// TIA Portal V20 export
TYPE "type_emRelations_em4_sequence"
// stored: Access Published, Namespace Unit1
   STRUCT
      sideTapeLoading : Struct
         jobs : "LAF_typeJobs";
         sequence : "LAF_typeSequence";
         selectJobStatus { S7_SetPoint := 'True'} : Array[0..10] of "LAF_typeJobStatus";
         "step" : "LER_typeStep";
         jobInterface : Struct
            chargeJob2 : "LER_typeJobInterface";
         END_STRUCT;
         homeCheck : Struct
            TapeLoadReq { ExternalWritable := 'False'} : Bool;
            TapeLoaded { ExternalWritable := 'False'} : Bool;
         END_STRUCT;
      END_STRUCT;
      sideTapeAttachment : Struct
         jobs : "LAF_typeJobs";
         sequence : "LAF_typeSequence";
         selectJobStatus { S7_SetPoint := 'True'} : Array[0..10] of "LAF_typeJobStatus";
         "step" : "LER_typeStep";
         jobInterface : Struct
            rightTapeGetJob2 : "LER_typeJobInterface";
            leftTapeGetJob3 : "LER_typeJobInterface";
            tape1PutJob4 : "LER_typeJobInterface";
            tape2PutJob5 : "LER_typeJobInterface";
            tape3PutJob6 : "LER_typeJobInterface";
            tape4PutJob7 : "LER_typeJobInterface";
            TapeIdleJob8 { S7_SetPoint := 'True'} : "LER_typeJobInterface";
         END_STRUCT;
         homeCheck : Struct
            waitPosTapeGetReq { ExternalWritable := 'False'} : Bool;
            waitPosTapeLeftGet { ExternalWritable := 'False'} : Bool;
            waitPosTapeRightGet { ExternalWritable := 'False'} : Bool;
            waitPosTapeAllGet { ExternalWritable := 'False'} : Bool;
            putPosTapeAllGet { ExternalWritable := 'False'} : Bool;
         END_STRUCT;
      END_STRUCT;
      sideTapeFixStage : Struct
         jobs : "LAF_typeJobs";
         sequence : "LAF_typeSequence";
         selectJobStatus { S7_SetPoint := 'True'} : Array[0..10] of "LAF_typeJobStatus";
         "step" : "LER_typeStep";
         jobInterface : Struct
            loadJob2 : "LER_typeJobInterface";
            taping1Job3 : "LER_typeJobInterface";
            taping2Job4 : "LER_typeJobInterface";
            taping3Job5 : "LER_typeJobInterface";
            taping4Job6 : "LER_typeJobInterface";
            unloadJob7 : "LER_typeJobInterface";
         END_STRUCT;
         homeCheck : Struct
            tape1PosPartNoDetect { ExternalWritable := 'False'} : Bool;
            tape1PosPartDetect { ExternalWritable := 'False'} : Bool;
            tape2PosPartDetect { ExternalWritable := 'False'} : Bool;
            tape3PosPartDetect { ExternalWritable := 'False'} : Bool;
            tape4PosPartDetect { ExternalWritable := 'False'} : Bool;
         END_STRUCT;
      END_STRUCT;
   END_STRUCT;
   // // sideTapeLoading."step".action1[101] : Step[101] : JOB[1] Condition
   // // sideTapeLoading."step".action1[110] : Step[110] : Side Tape Loading Down
   // // sideTapeLoading."step".action1[120] : Step[120] : Side Tape Clamp Open
   // // sideTapeLoading."step".action1[130] : Step[130] : Side Tape Cutter Backward
   // // sideTapeLoading."step".action1[140] : Step[140] : Side Tape Cutter Clamp Forward
   // // sideTapeLoading."step".action1[150] : Step[150] : Side Tape Tension Backward
   // // sideTapeLoading."step".action1[190] : Step[190] : JOB[1] Step End
   // // sideTapeLoading."step".action1[201] : Step[201] : JOB[2] Condition
   // // sideTapeLoading."step".action1[210] : Step[210] : Side Tape Loading Up, Tension Backward
   // // sideTapeLoading."step".action1[220] : Step[220] : Side Tape Clamp Close
   // // sideTapeLoading."step".action1[230] : Step[230] : Side Tape Cutter Clamp Backward
   // // sideTapeLoading."step".action1[240] : Step[240] : Side Tape Loading Down, Tension Forward
   // // sideTapeLoading."step".action1[250] : Step[250] : Side Tape Cutter Clamp Forward
   // // sideTapeLoading."step".action1[260] : Step[260] : Side Tape Tension Backward
   // // sideTapeLoading."step".action1[290] : Step[290] : JOB[2] Step End
   // // sideTapeLoading."step".transition1[101] : Step[101] : JOB[1] Condition
   // // sideTapeLoading."step".transition1[110] : Step[110] : Side Tape Loading Down
   // // sideTapeLoading."step".transition1[120] : Step[120] : Side Tape Clamp Open
   // // sideTapeLoading."step".transition1[130] : Step[130] : Side Tape Cutter Backward
   // // sideTapeLoading."step".transition1[140] : Step[140] : Side Tape Cutter Clamp Forward
   // // sideTapeLoading."step".transition1[150] : Step[150] : Side Tape Tension Backward
   // // sideTapeLoading."step".transition1[190] : Step[190] : JOB[1] Step End
   // // sideTapeLoading."step".transition1[201] : Step[201] : JOB[2] Condition
   // // sideTapeLoading."step".transition1[210] : Step[210] : Side Tape Loading Up, Tension Backward
   // // sideTapeLoading."step".transition1[220] : Step[220] : Side Tape Clamp Close
   // // sideTapeLoading."step".transition1[230] : Step[230] : Side Tape Cutter Clamp Backward
   // // sideTapeLoading."step".transition1[240] : Step[240] : Side Tape Loading Down, Tension Forward
   // // sideTapeLoading."step".transition1[250] : Step[250] : Side Tape Cutter Clamp Forward
   // // sideTapeLoading."step".transition1[260] : Step[260] : Side Tape Tension Backward
   // // sideTapeLoading."step".transition1[290] : Step[290] : JOB[2] Step End
   // // sideTapeAttachment."step".action1[101] : Step[101] : JOB[1] Condition
   // // sideTapeAttachment."step".action1[110] : Step[110] : Side Tape Attachment Left, Right Backward
   // // sideTapeAttachment."step".action1[111] : Step[111] : Side Tape Attachment Y-Axis Wait Pos
   // // sideTapeAttachment."step".action1[120] : Step[120] : Side Tape Attachment Bottom Forward
   // // sideTapeAttachment."step".action1[130] : Step[130] : Side Tape Attachment Remain Attach Left Condition
   // // sideTapeAttachment."step".action1[131] : Step[131] : Side Tape Attachment X-Axis Remain Attach Left Position
   // // sideTapeAttachment."step".action1[132] : Step[132] : Side Tape Attachment Y-Axis Remain Attach Left Position
   // // sideTapeAttachment."step".action1[133] : Step[133] : Side Tape Attachment Left Vaccum Off
   // // sideTapeAttachment."step".action1[134] : Step[134] : Side Tape Attachment Y-Axis Wait Pos
   // // sideTapeAttachment."step".action1[140] : Step[140] : Side Tape Attachment Remain Attach Right Condition
   // // sideTapeAttachment."step".action1[141] : Step[141] : Side Tape Attachment X-Axis Remain Attach Right Position
   // // sideTapeAttachment."step".action1[142] : Step[142] : Side Tape Attachment Y-Axis Remain Attach Right Position
   // // sideTapeAttachment."step".action1[143] : Step[143] : Side Tape Attachment Right Vaccum Off
   // // sideTapeAttachment."step".action1[144] : Step[144] : Side Tape Attachment Y-Axis Wait Pos
   // // sideTapeAttachment."step".action1[180] : Step[180] : Side Tape Attachment X-Axis Wait Position
   // // sideTapeAttachment."step".action1[190] : Step[190] : Job[1] Step End
   // // sideTapeAttachment."step".action1[201] : Step[201] : JOB[2] Condition
   // // sideTapeAttachment."step".action1[210] : Step[210] : Side Tape Attachment X-Axis Right Loading Pos
   // // sideTapeAttachment."step".action1[220] : Step[220] : Side Tape Attachment Y-Axis Loading Pos
   // // sideTapeAttachment."step".action1[221] : Step[221] : Side Tape Attachment-2 Vaccum On
   // // sideTapeAttachment."step".action1[230] : Step[230] : Side Tape Cutter Forward
   // // sideTapeAttachment."step".action1[231] : Step[231] : Side Tape Cutter Backward
   // // sideTapeAttachment."step".action1[240] : Step[240] : Side Tape Clamp Open
   // // sideTapeAttachment."step".action1[241] : Step[241] : Spare
   // // sideTapeAttachment."step".action1[270] : Step[270] : Side Tape Attachment Y-Axis Wait Pos
   // // sideTapeAttachment."step".action1[280] : Step[280] : Side Tape Attachment X-Axis Wait Pos
   // // sideTapeAttachment."step".action1[290] : Step[290] : Job[2] Step End
   // // sideTapeAttachment."step".action1[301] : Step[301] : JOB[3] Condition
   // // sideTapeAttachment."step".action1[310] : Step[310] : Side Tape Attachment X-Axis Left Loading Pos
   // // sideTapeAttachment."step".action1[320] : Step[320] : Side Tape Attachment Y-Axis Loading Pos
   // // sideTapeAttachment."step".action1[321] : Step[321] : Side Tape Attachment-1 Vaccum On
   // // sideTapeAttachment."step".action1[330] : Step[330] : Side Tape Cutter Forward
   // // sideTapeAttachment."step".action1[331] : Step[331] : Side Tape Cutter Backward
   // // sideTapeAttachment."step".action1[340] : Step[340] : Side Tape Clamp Open
   // // sideTapeAttachment."step".action1[341] : Step[341] : Spare
   // // sideTapeAttachment."step".action1[370] : Step[370] : Side Tape Attachment Y-Axis Wait Pos
   // // sideTapeAttachment."step".action1[380] : Step[380] : Side Tape Attachment X-Axis Tape-1 Put Pos
   // // sideTapeAttachment."step".action1[390] : Step[390] : Job[3] Step End
   // // sideTapeAttachment."step".action1[401] : Step[401] : JOB[4] Condition
   // // sideTapeAttachment."step".action1[410] : Step[410] : Side Tape Attachment X-Axis Tape-1 Put Pos
   // // sideTapeAttachment."step".action1[420] : Step[420] : Side tape Attachment Y-Axis Tape-1 Put Pos
   // // sideTapeAttachment."step".action1[421] : Step[421] : Side Tape Attachment Left, Right Forward, Vaccum Off
   // // sideTapeAttachment."step".action1[422] : Step[422] : Spare
   // // sideTapeAttachment."step".action1[430] : Step[430] : Side Tape Attachment Left, Right Backward
   // // sideTapeAttachment."step".action1[431] : Step[431] : Side Tape Attachment Y-Axis Wait Pos
   // // sideTapeAttachment."step".action1[480] : Step[480] : Side Tape Attachment X-Axis Wait Pos
   // // sideTapeAttachment."step".action1[490] : Step[490] : Job[4] Step End
   // // sideTapeAttachment."step".action1[501] : Step[501] : Job[5] Condition
   // // sideTapeAttachment."step".action1[510] : Step[510] : Side Tape Attachment X-Axis Tape-2 Put Pos
   // // sideTapeAttachment."step".action1[520] : Step[520] : Side tape Attachment Y-Axis Tape-2 Put Pos
   // // sideTapeAttachment."step".action1[521] : Step[521] : Side Tape Attachment Right Forward, Vaccum Off
   // // sideTapeAttachment."step".action1[522] : Step[522] : Spare
   // // sideTapeAttachment."step".action1[530] : Step[530] : Side Tape Attachment Right Backward
   // // sideTapeAttachment."step".action1[531] : Step[531] : Side Tape Attachment Y-Axis Wait Pos
   // // sideTapeAttachment."step".action1[580] : Step[580] : Side Tape Attachment X-Axis Wait Pos
   // // sideTapeAttachment."step".action1[590] : Step[590] : Job[5] Step End
   // // sideTapeAttachment."step".action1[601] : Step[601] : Job[6] Condition
   // // sideTapeAttachment."step".action1[610] : Step[610] : Side Tape Attachment X-Axis Tape-3 Put Pos
   // // sideTapeAttachment."step".action1[620] : Step[620] : Side tape Attachment Y-Axis Tape-2 Put Pos
   // // sideTapeAttachment."step".action1[621] : Step[621] : Side Tape Attachment Right Forward, Vaccum Off
   // // sideTapeAttachment."step".action1[622] : Step[622] : Spare
   // // sideTapeAttachment."step".action1[630] : Step[630] : Side Tape Attachment Right Backward
   // // sideTapeAttachment."step".action1[631] : Step[631] : Side Tape Attachment Y-Axis Wait Pos
   // // sideTapeAttachment."step".action1[680] : Step[680] : Side Tape Attachment X-Axis Wait Pos
   // // sideTapeAttachment."step".action1[690] : Step[690] : Job[6] Step End
   // // sideTapeAttachment."step".action1[701] : Step[701] : Job[7] Condition
   // // sideTapeAttachment."step".action1[710] : Step[710] : Side Tape Attachment X-Axis Tape-4 Put Pos
   // // sideTapeAttachment."step".action1[720] : Step[720] : Side tape Attachment Y-Axis Tape-1 Put Pos
   // // sideTapeAttachment."step".action1[721] : Step[721] : Side Tape Attachment Right Forward, Vaccum Off
   // // sideTapeAttachment."step".action1[722] : Step[722] : Spare
   // // sideTapeAttachment."step".action1[730] : Step[730] : Side Tape Attachment Right Backward
   // // sideTapeAttachment."step".action1[731] : Step[731] : Side Tape Attachment Y-Axis Wait Pos
   // // sideTapeAttachment."step".action1[780] : Step[780] : Side Tape Attachment X-Axis Wait Pos
   // // sideTapeAttachment."step".action1[790] : Step[790] : Job[7] Step End
   // // sideTapeAttachment."step".transition1[101] : Step[101] : JOB[1] Condition
   // // sideTapeAttachment."step".transition1[110] : Step[110] : Side Tape Attachment Left, Right Backward
   // // sideTapeAttachment."step".transition1[111] : Step[111] : Side Tape Attachment Y-Axis Wait Pos
   // // sideTapeAttachment."step".transition1[180] : Step[180] : Side Tape Attachment Bottom Forward
   // // sideTapeAttachment."step".transition1[181] : Step[181] : Side Tape Attachment X-Axis Wait Position
   // // sideTapeAttachment."step".transition1[190] : Step[190] : Job[1] Step End
   // // sideTapeAttachment."step".transition1[201] : Step[201] : JOB[2] Condition
   // // sideTapeAttachment."step".transition1[210] : Step[210] : Side Tape Attachment X-Axis Right Loading Pos
   // // sideTapeAttachment."step".transition1[220] : Step[220] : Side Tape Attachment Y-Axis Loading Pos
   // // sideTapeAttachment."step".transition1[221] : Step[221] : Side Tape Attachment-2 Vaccum On
   // // sideTapeAttachment."step".transition1[230] : Step[230] : Side Tape Cutter Forward
   // // sideTapeAttachment."step".transition1[231] : Step[231] : Side Tape Cutter Backward
   // // sideTapeAttachment."step".transition1[240] : Step[240] : Side Tape Clamp Open
   // // sideTapeAttachment."step".transition1[241] : Step[241] : Spare
   // // sideTapeAttachment."step".transition1[270] : Step[270] : Side Tape Attachment Y-Axis Wait Pos
   // // sideTapeAttachment."step".transition1[280] : Step[280] : Side Tape Attachment X-Axis Wait Pos
   // // sideTapeAttachment."step".transition1[290] : Step[290] : Job[2] Step End
   // // sideTapeAttachment."step".transition1[301] : Step[301] : JOB[3] Condition
   // // sideTapeAttachment."step".transition1[310] : Step[310] : Side Tape Attachment X-Axis Left Loading Pos
   // // sideTapeAttachment."step".transition1[320] : Step[320] : Side Tape Attachment Y-Axis Loading Pos
   // // sideTapeAttachment."step".transition1[321] : Step[321] : Side Tape Attachment-1 Vaccum On
   // // sideTapeAttachment."step".transition1[330] : Step[330] : Side Tape Cutter Forward
   // // sideTapeAttachment."step".transition1[331] : Step[331] : Side Tape Cutter Backward
   // // sideTapeAttachment."step".transition1[340] : Step[340] : Side Tape Clamp Open
   // // sideTapeAttachment."step".transition1[341] : Step[341] : Spare
   // // sideTapeAttachment."step".transition1[370] : Step[370] : Side Tape Attachment Y-Axis Wait Pos
   // // sideTapeAttachment."step".transition1[380] : Step[380] : Side Tape Attachment X-Axis Tape-1 Put Pos
   // // sideTapeAttachment."step".transition1[390] : Step[390] : Job[3] Step End
   // // sideTapeAttachment."step".transition1[401] : Step[401] : JOB[4] Condition
   // // sideTapeAttachment."step".transition1[410] : Step[410] : Side Tape Attachment X-Axis Tape-1 Put Pos
   // // sideTapeAttachment."step".transition1[420] : Step[420] : Side tape Attachment Y-Axis Tape-1 Put Pos
   // // sideTapeAttachment."step".transition1[421] : Step[421] : Side Tape Attachment Left, Right Forward, Vaccum Off
   // // sideTapeAttachment."step".transition1[422] : Step[422] : Spare
   // // sideTapeAttachment."step".transition1[430] : Step[430] : Side Tape Attachment Left, Right Backward
   // // sideTapeAttachment."step".transition1[431] : Step[431] : Side Tape Attachment Y-Axis Wait Pos
   // // sideTapeAttachment."step".transition1[480] : Step[480] : Side Tape Attachment X-Axis Wait Pos
   // // sideTapeAttachment."step".transition1[490] : Step[490] : Job[4] Step End
   // // sideTapeAttachment."step".transition1[501] : Step[501] : Job[5] Condition
   // // sideTapeAttachment."step".transition1[510] : Step[510] : Side Tape Attachment X-Axis Tape-2 Put Pos
   // // sideTapeAttachment."step".transition1[520] : Step[520] : Side tape Attachment Y-Axis Tape-2 Put Pos
   // // sideTapeAttachment."step".transition1[521] : Step[521] : Side Tape Attachment Right Forward, Vaccum Off
   // // sideTapeAttachment."step".transition1[522] : Step[522] : Spare
   // // sideTapeAttachment."step".transition1[530] : Step[530] : Side Tape Attachment Right Backward
   // // sideTapeAttachment."step".transition1[531] : Step[531] : Side Tape Attachment Y-Axis Wait Pos
   // // sideTapeAttachment."step".transition1[580] : Step[580] : Side Tape Attachment X-Axis Wait Pos
   // // sideTapeAttachment."step".transition1[590] : Step[590] : Job[5] Step End
   // // sideTapeAttachment."step".transition1[601] : Step[601] : Job[6] Condition
   // // sideTapeAttachment."step".transition1[610] : Step[610] : Side Tape Attachment X-Axis Tape-3 Put Pos
   // // sideTapeAttachment."step".transition1[620] : Step[620] : Side tape Attachment Y-Axis Tape-2 Put Pos
   // // sideTapeAttachment."step".transition1[621] : Step[621] : Side Tape Attachment Right Forward, Vaccum Off
   // // sideTapeAttachment."step".transition1[622] : Step[622] : Spare
   // // sideTapeAttachment."step".transition1[630] : Step[630] : Side Tape Attachment Right Backward
   // // sideTapeAttachment."step".transition1[631] : Step[631] : Side Tape Attachment Y-Axis Wait Pos
   // // sideTapeAttachment."step".transition1[680] : Step[680] : Side Tape Attachment X-Axis Wait Pos
   // // sideTapeAttachment."step".transition1[690] : Step[690] : Job[6] Step End
   // // sideTapeAttachment."step".transition1[701] : Step[701] : Job[7] Condition
   // // sideTapeAttachment."step".transition1[710] : Step[710] : Side Tape Attachment X-Axis Tape-4 Put Pos
   // // sideTapeAttachment."step".transition1[720] : Step[720] : Side tape Attachment Y-Axis Tape-1 Put Pos
   // // sideTapeAttachment."step".transition1[721] : Step[721] : Side Tape Attachment Right Forward, Vaccum Off
   // // sideTapeAttachment."step".transition1[722] : Step[722] : Spare
   // // sideTapeAttachment."step".transition1[730] : Step[730] : Side Tape Attachment Right Backward
   // // sideTapeAttachment."step".transition1[731] : Step[731] : Side Tape Attachment Y-Axis Wait Pos
   // // sideTapeAttachment."step".transition1[780] : Step[780] : Side Tape Attachment X-Axis Wait Pos
   // // sideTapeAttachment."step".transition1[790] : Step[790] : Job[7] Step End
   // // sideTapeFixStage."step".action1[101] : Step[101] : JOB[1] Condition
   // // sideTapeFixStage."step".action1[110] : Step[110] : Side Tape Fix Stage Clamp Open
   // // sideTapeFixStage."step".action1[111] : Step[111] : Side Tape Fix Stage Clamp Close
   // // sideTapeFixStage."step".action1[120] : Step[120] : Side Tape Fix Stage X-Axis JR Get Pos
   // // sideTapeFixStage."step".action1[130] : Step[130] : Side Tape Fix Stage C-Axis Wait Pos [Tape-1]
   // // sideTapeFixStage."step".action1[131] : Step[131] : Side Tape Fix Stage C-Axis Tape-2 Pos
   // // sideTapeFixStage."step".action1[132] : Step[132] : Side Tape Fix Stage C-Axis Tape-3 Pos
   // // sideTapeFixStage."step".action1[133] : Step[133] : Side Tape Fix Stage C-Axis Tape-4 Pos
   // // sideTapeFixStage."step".action1[140] : Step[140] : Side Tape Fix Stage X-Axis Wait Pos
   // // sideTapeFixStage."step".action1[190] : Step[190] : JOB[1] Step End
   // // sideTapeFixStage."step".action1[201] : Step[201] : JOB[2] Condition
   // // sideTapeFixStage."step".action1[210] : Step[210] : Side Tape Fix Stage [Loading Request] => JR PP Right
   // // sideTapeFixStage."step".action1[220] : Step[220] : Side Tape Fix Stage X-Axis JR Get Pos
   // // sideTapeFixStage."step".action1[230] : Step[230] : Side Tape Fix Stage Clamp Close
   // // sideTapeFixStage."step".action1[231] : Step[231] : Data Transfer
   // // sideTapeFixStage."step".action1[232] : Step[232] : Side Tape Fix Stage [Unclamp Request] => JR PP Right
   // // sideTapeFixStage."step".action1[280] : Step[280] : Side Tape Fix Stage X-Axis Wait Pos
   // // sideTapeFixStage."step".action1[290] : Step[290] : JOB[2] Step End
   // // sideTapeFixStage."step".action1[301] : Step[301] : JOB[4] Condition
   // // sideTapeFixStage."step".action1[310] : Step[310] : Spare
   // // sideTapeFixStage."step".action1[320] : Step[320] : Side Tape Fix Stage => Call Attachment Tape-1
   // // sideTapeFixStage."step".action1[390] : Step[390] : JOB[3] Step End
   // // sideTapeFixStage."step".action1[401] : Step[401] : JOB[4] Condition
   // // sideTapeFixStage."step".action1[410] : Step[410] : Side Tape Fix Stage X-Axis Wait Pos
   // // sideTapeFixStage."step".action1[411] : Step[411] : Side Tape Fix Stage C-Axis Taping-2 Pos
   // // sideTapeFixStage."step".action1[412] : Step[412] : Side Tape Fix Stage X-Axis Wait Pos
   // // sideTapeFixStage."step".action1[420] : Step[420] : Side Tape Fix Stage => Call Attachment Tape-2
   // // sideTapeFixStage."step".action1[490] : Step[490] : JOB[4] Step End
   // // sideTapeFixStage."step".action1[501] : Step[501] : JOB[5] Condition
   // // sideTapeFixStage."step".action1[510] : Step[510] : Side Tape Fix Stage X-Axis Wait Pos
   // // sideTapeFixStage."step".action1[511] : Step[511] : Side Tape Fix Stage C-Axis Taping-3 Pos
   // // sideTapeFixStage."step".action1[512] : Step[512] : Side Tape Fix Stage X-Axis Wait Pos
   // // sideTapeFixStage."step".action1[520] : Step[520] : Side Tape Fix Stage => Call Attachment Tape-3
   // // sideTapeFixStage."step".action1[590] : Step[590] : JOB[5] Step End
   // // sideTapeFixStage."step".action1[601] : Step[601] : JOB[6] Condition
   // // sideTapeFixStage."step".action1[610] : Step[610] : Side Tape Fix Stage X-Axis Wait Pos
   // // sideTapeFixStage."step".action1[611] : Step[611] : Side Tape Fix Stage C-Axis Taping-4 Pos
   // // sideTapeFixStage."step".action1[612] : Step[612] : Side Tape Fix Stage X-Axis Wait Pos
   // // sideTapeFixStage."step".action1[620] : Step[620] : Side Tape Fix Stage => Call Attachment Tape-4
   // // sideTapeFixStage."step".action1[690] : Step[690] : JOB[6] Step End
   // // sideTapeFixStage."step".action1[701] : Step[701] : JOB[7] Condition
   // // sideTapeFixStage."step".action1[710] : Step[710] : Side Tape Fix Stage X-Axis Put Pos
   // // sideTapeFixStage."step".action1[720] : Step[720] : Side Tape Fix Stage [Unloading Request] => Transfer PP Left
   // // sideTapeFixStage."step".action1[721] : Step[721] : Side Tape Fix Stage [Clamp Request] => Transfer PP Left
   // // sideTapeFixStage."step".action1[722] : Step[722] : Side Tape Fix Stage Clamp Open
   // // sideTapeFixStage."step".action1[723] : Step[723] : Side Tape Fix Stage [Backward Request] => Transfer PP Left
   // // sideTapeFixStage."step".action1[780] : Step[780] : Side Tape Fix Stage X-Axis Wait Pos
   // // sideTapeFixStage."step".action1[781] : Step[781] : Side Tape Fix Stage C-Axis Wait Pos
   // // sideTapeFixStage."step".action1[782] : Step[782] : Side Tape Fix Stage X-Axis Wait Pos
   // // sideTapeFixStage."step".action1[790] : Step[790] : JOB[7] Step End
   // // sideTapeFixStage."step".transition1[101] : Step[101] : JOB[1] Condition
   // // sideTapeFixStage."step".transition1[110] : Step[110] : Side Tape Fix Stage Clamp Open
   // // sideTapeFixStage."step".transition1[111] : Step[111] : Side Tape Fix Stage Clamp Close
   // // sideTapeFixStage."step".transition1[120] : Step[120] : Side Tape Fix Stage X-Axis JR Get Pos
   // // sideTapeFixStage."step".transition1[130] : Step[130] : Side Tape Fix Stage C-Axis Wait Pos [Tape-1]
   // // sideTapeFixStage."step".transition1[131] : Step[131] : Side Tape Fix Stage C-Axis Tape-2 Pos
   // // sideTapeFixStage."step".transition1[132] : Step[132] : Side Tape Fix Stage C-Axis Tape-3 Pos
   // // sideTapeFixStage."step".transition1[133] : Step[133] : Side Tape Fix Stage C-Axis Tape-4 Pos
   // // sideTapeFixStage."step".transition1[140] : Step[140] : Side Tape Fix Stage X-Axis Wait Pos
   // // sideTapeFixStage."step".transition1[190] : Step[190] : JOB[1] Step End
   // // sideTapeFixStage."step".transition1[201] : Step[201] : JOB[2] Condition
   // // sideTapeFixStage."step".transition1[210] : Step[210] : Side Tape Fix Stage [Loading Request] => JR PP Right
   // // sideTapeFixStage."step".transition1[220] : Step[220] : Side Tape Fix Stage X-Axis JR Get Pos
   // // sideTapeFixStage."step".transition1[230] : Step[230] : Side Tape Fix Stage Clamp Close
   // // sideTapeFixStage."step".transition1[231] : Step[231] : Data Transfer
   // // sideTapeFixStage."step".transition1[232] : Step[232] : Side Tape Fix Stage [Unclamp Request] => JR PP Right
   // // sideTapeFixStage."step".transition1[280] : Step[280] : Side Tape Fix Stage X-Axis Wait Pos
   // // sideTapeFixStage."step".transition1[290] : Step[290] : JOB[2] Step End
   // // sideTapeFixStage."step".transition1[301] : Step[301] : JOB[4] Condition
   // // sideTapeFixStage."step".transition1[310] : Step[310] : Spare
   // // sideTapeFixStage."step".transition1[320] : Step[320] : Side Tape Fix Stage => Call Attachment Tape-1
   // // sideTapeFixStage."step".transition1[390] : Step[390] : JOB[3] Step End
   // // sideTapeFixStage."step".transition1[401] : Step[401] : JOB[4] Condition
   // // sideTapeFixStage."step".transition1[410] : Step[410] : Side Tape Fix Stage X-Axis Wait Pos
   // // sideTapeFixStage."step".transition1[411] : Step[411] : Side Tape Fix Stage C-Axis Taping-2 Pos
   // // sideTapeFixStage."step".transition1[412] : Step[412] : Side Tape Fix Stage X-Axis Wait Pos
   // // sideTapeFixStage."step".transition1[420] : Step[420] : Side Tape Fix Stage => Call Attachment Tape-2
   // // sideTapeFixStage."step".transition1[490] : Step[490] : JOB[4] Step End
   // // sideTapeFixStage."step".transition1[501] : Step[501] : JOB[5] Condition
   // // sideTapeFixStage."step".transition1[510] : Step[510] : Side Tape Fix Stage X-Axis Wait Pos
   // // sideTapeFixStage."step".transition1[511] : Step[511] : Side Tape Fix Stage C-Axis Taping-3 Pos
   // // sideTapeFixStage."step".transition1[512] : Step[512] : Side Tape Fix Stage X-Axis Wait Pos
   // // sideTapeFixStage."step".transition1[520] : Step[520] : Side Tape Fix Stage => Call Attachment Tape-3
   // // sideTapeFixStage."step".transition1[590] : Step[590] : JOB[5] Step End
   // // sideTapeFixStage."step".transition1[601] : Step[601] : JOB[6] Condition
   // // sideTapeFixStage."step".transition1[610] : Step[610] : Side Tape Fix Stage X-Axis Wait Pos
   // // sideTapeFixStage."step".transition1[611] : Step[611] : Side Tape Fix Stage C-Axis Taping-4 Pos
   // // sideTapeFixStage."step".transition1[612] : Step[612] : Side Tape Fix Stage X-Axis Wait Pos
   // // sideTapeFixStage."step".transition1[620] : Step[620] : Side Tape Fix Stage => Call Attachment Tape-4
   // // sideTapeFixStage."step".transition1[690] : Step[690] : JOB[6] Step End
   // // sideTapeFixStage."step".transition1[701] : Step[701] : JOB[7] Condition
   // // sideTapeFixStage."step".transition1[710] : Step[710] : Side Tape Fix Stage X-Axis Put Pos
   // // sideTapeFixStage."step".transition1[720] : Step[720] : Side Tape Fix Stage [Unloading Request] => Transfer PP Left
   // // sideTapeFixStage."step".transition1[721] : Step[721] : Side Tape Fix Stage [Clamp Request] => Transfer PP Left
   // // sideTapeFixStage."step".transition1[722] : Step[722] : Side Tape Fix Stage Clamp Open
   // // sideTapeFixStage."step".transition1[723] : Step[723] : Side Tape Fix Stage [Backward Request] => Transfer PP Left
   // // sideTapeFixStage."step".transition1[780] : Step[780] : Side Tape Fix Stage X-Axis Wait Pos
   // // sideTapeFixStage."step".transition1[781] : Step[781] : Side Tape Fix Stage C-Axis Wait Pos
   // // sideTapeFixStage."step".transition1[782] : Step[782] : Side Tape Fix Stage X-Axis Wait Pos
   // // sideTapeFixStage."step".transition1[790] : Step[790] : JOB[7] Step End
END_TYPE
